(* IEC 61131-3 sources: CodesysTest/alpha/export/FBs/Components/Motors/Applied Motion/FB_AppliedMotionStepServoTCP.pou, 2 files *)

(* ---- ExecuteStoredProgram.m.st ---- *)
(*#-#-#-#-#-#-#-#-#-#---Declaration---#-#-#-#-#-#-#-#-#-#-#-#-#*)

METHOD ExecuteStoredProgram
VAR_INPUT
    (*Program number to execute*)
    programNumber    : INT;
END_VAR
(*#-#-#-#-#-#-#-#-#-#---Implementation---#-#-#-#-#-#-#-#-#-#-#-#-#*)

//Load program into queue by setting it as parameter 1 and send it and the execute queue opcode
commandSuccessful := FALSE;
SendOpcodeCommand.opcode := STEP_SERVO_OPCODES.QUEUE_LOAD_AND_EXECUTE;
SendOpcodeCommand.Parameter1 := INT_TO_WORD(programNumber);
SendOpcodeCommand.Execute();

(* ---- MoveDistance.m.st ---- *)
(*#-#-#-#-#-#-#-#-#-#---Declaration---#-#-#-#-#-#-#-#-#-#-#-#-#*)

METHOD MoveDistance
VAR_INPUT
    distance : REAL;        //Distance to move in inches
    acceleration : INT;        //Acceleration in RPM/sec
    deceleration : INT;        //Deceleration in RPM/sec
    velocity : INT;            //Velocity in .25RPM
END_VAR(*#-#-#-#-#-#-#-#-#-#---Implementation---#-#-#-#-#-#-#-#-#-#-#-#-#*)

//This method preps the data to send to the drive and triggers the send.
//Set distance and unpack to prep data to send to motor
distanceToMoveInSteps.rawValue := REAL_TO_DINT((distance) * stepsPerInchSetpoint);
IF reversePolarity THEN
    distanceToMoveInSteps.rawValue := distanceToMoveInSteps.rawValue * -1;
END_IF
commandSuccessful := FALSE;
ModbusLongHandler.Unpack(distanceToMoveInSteps);
sendMoveCommand.acceleration := acceleration;
sendMoveCommand.deceleration := deceleration;
sendMoveCommand.velocity := velocity;
sendMoveCommand.distanceHighWord := distanceToMoveInSteps.highWord;
sendMoveCommand.distanceLowWord := distanceToMoveInSteps.lowWord;
sendMoveCommand.opcode := STEP_SERVO_OPCODES.FEED_TO_LENGTH;
sendMoveCommand.Execute();
